// TIA Portal V17 export
// export: Created 2022-10-14T12:26:44.1091034Z, ExportSetting WithDefaults, DisplayName Totally Integrated Automation Portal, DisplayVersion V17 Update 4, DisplayName TIA Portal Openness, DisplayVersion V17 Update 4, DisplayName TIA Portal Version Control Interface, DisplayVersion V17, DisplayName SINAMICS Startdrive Advanced, DisplayVersion V17 Update2, DisplayName SINAMICS Startdrive G130, G150, S120, S150, SINAMICS MV, S210, DisplayVersion V17 Update2, DisplayName SINAMICS Startdrive G110M, G120, G120C, G120D, G120P, G115D, DisplayVersion V17 Update2, DisplayName STEP 7 Professional, DisplayVersion V17 Update 4, DisplayName STEP 7 Safety, DisplayVersion V17, DisplayName WinCC Advanced / Unified PC, DisplayVersion V17 Update 4
DATA_BLOCK "2000_Data"   // DB2000
{ S7_Optimized_Access := 'TRUE' }
VERSION : 0.1
// stored: AutoNumber false, DBAccessibleFromOPCUA true, DBAccessibleFromWebserver true, IsOnlyStoredInLoadMemory false, IsRetainMemResEnabled false, IsWriteProtectedInAS false, MemoryReserve 100
   VAR
      Addr : Array[1.."DeviceNr"] of Byte;
      Gruppen { S7_SetPoint := 'True'} : Array[1.."DeviceNr"] of "Channels";
      Devices_Data : Array[1.."DeviceNr"] of "Dates_Pro_Channel";
   END_VAR
BEGIN
   Addr[1] := 16#02;
   Addr[2] := 16#03;
   Addr[3] := 16#04;
   Addr[4..6] := 16#05;
   Gruppen[1].Kanal[1] := 16#01;
   Gruppen[1].Kanal[2] := 16#02;
   Gruppen[1].Kanal[3] := 16#03;
   Gruppen[1].Kanal[4] := 16#04;
   Gruppen[2].Kanal[1] := 16#01;
   Gruppen[2].Kanal[2] := 16#02;
   Gruppen[2].Kanal[3] := 16#03;
   Gruppen[2].Kanal[4] := 16#04;
   Gruppen[3].Kanal[1] := 16#01;
   Gruppen[3].Kanal[2] := 16#02;
   Gruppen[3].Kanal[3] := 16#03;
   Gruppen[3].Kanal[4] := 16#04;
   Gruppen[4].Kanal[1] := 16#01;
   Gruppen[4].Kanal[2] := 16#02;
   Gruppen[4].Kanal[3] := 16#03;
   Gruppen[4].Kanal[4] := 16#04;
   Gruppen[5].Kanal[1] := 16#05;
   Gruppen[5].Kanal[2] := 16#06;
   Gruppen[5].Kanal[3] := 16#07;
   Gruppen[5].Kanal[4] := 16#08;
   Gruppen[6].Kanal[1] := 16#09;
   Gruppen[6].Kanal[2] := 16#0a;
   Gruppen[6].Kanal[3] := 16#0b;
   Gruppen[6].Kanal[4] := 16#0c;
END_DATA_BLOCK
